Omron CX-Programmer project NewProject (CX-Programmer 9.73)

# PLC NewPLC1: CP1E N30

## Global symbols (name address type ; comment)
100.00 BOOL  ; C MERAH
100.01 BOOL  ; C MERAH BELOK
100.02 BOOL  ; B MERAH
100.03 BOOL  ; B MERAH BELOK
100.04 BOOL  ; D MERAH
100.05 BOOL  ; D MERAH BELOK
100.06 BOOL  ; D KUNING
100.07 BOOL  ; D KUNING BELOK
100.08 BOOL  ; ;
100.09 BOOL  ; A HIJAU BELOK
100.10 BOOL  ; A KUNING BELOK
100.11 BOOL  ; C KUNING
100.12 BOOL  ; C HIJAU
100.13 BOOL  ; C KUNING BELOK
100.14 BOOL  ; C HIJAU BELOK
100.15 BOOL  ; B KUNING
101.00 BOOL  ; B KUNING BELOK
101.01 BOOL  ; B HIJAU
101.02 BOOL  ; B HIJAU BELOK
101.03 BOOL  ; D HIJAU BELOK
101.04 BOOL  ; D HIJAU
101.05 BOOL  ; A KUNING
101.06 BOOL  ; A MERAH
101.07 BOOL  ; A MERAH BELOK
101.08 BOOL  ; A HIJAU KEDIP
101.09 BOOL  ; B HIJAU KEDIP
101.10 BOOL  ; C HIJAU KEDIP
101.11 BOOL  ; D HIJAU KEDIP
102.00 BOOL  ; A KEDIP
102.01 BOOL  ; B KEDIP
102.02 BOOL  ; C KEDIP
102.03 BOOL  ; D KEDIP

## Program NewProgram1 (cyclic task 0)

### Section Section1

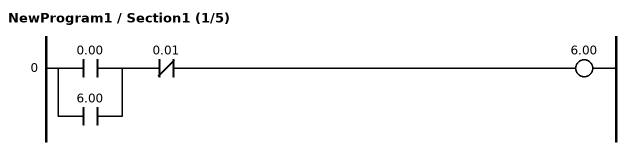
; rung 0
LD 0.00
OR 6.00
ANDNOT 0.01
OUT 6.00

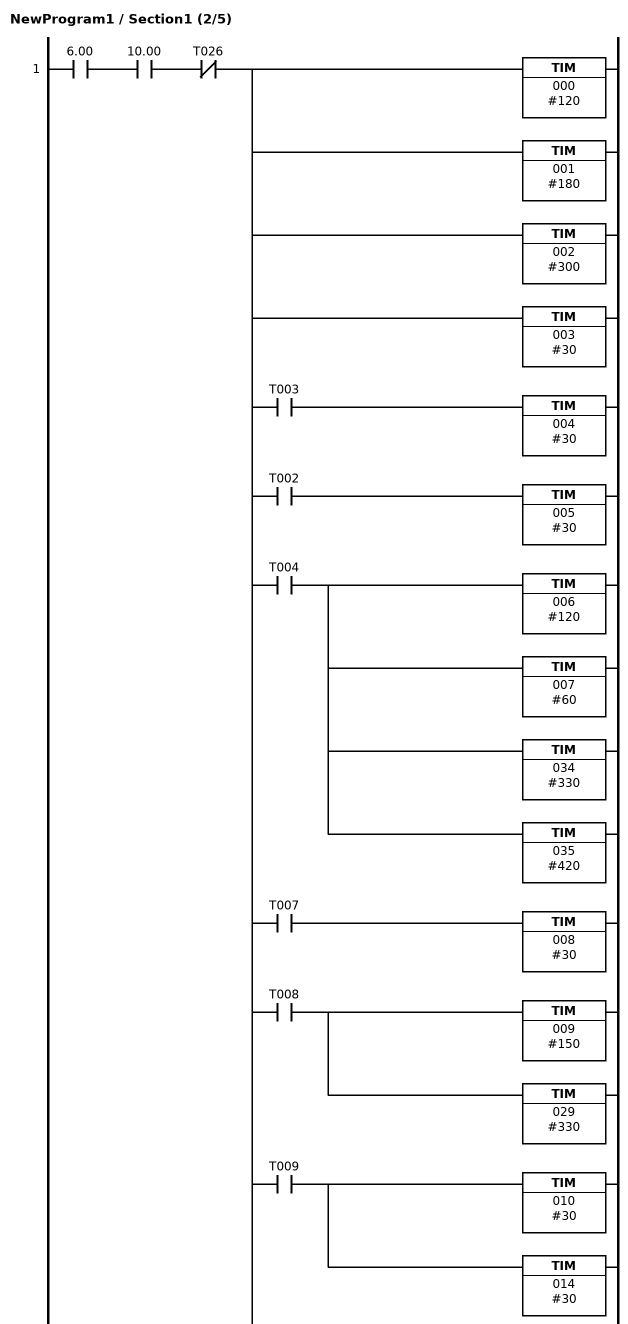

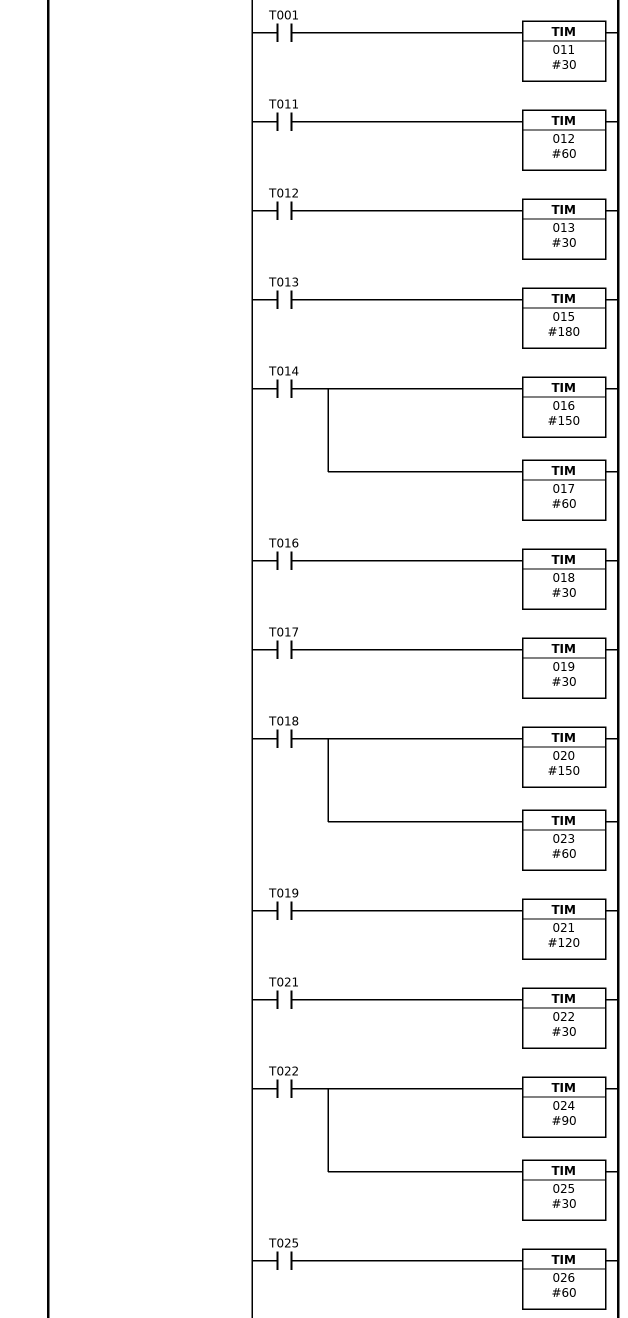

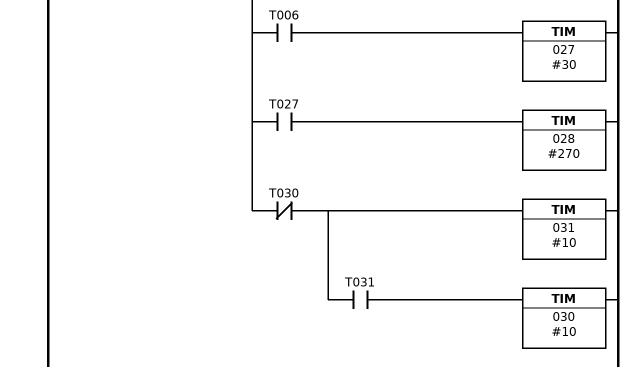
; rung 1
LD 6.00
AND 10.00
ANDNOT T026
OUT TR0
TIM 000 #120
TIM 001 #180
TIM 002 #300
TIM 003 #30
AND T003
TIM 004 #30
LD TR0
AND T002
TIM 005 #30
LD TR0
AND T004
TIM 006 #120
TIM 007 #60
TIM 034 #330
TIM 035 #420
LD TR0
AND T007
TIM 008 #30
LD TR0
AND T008
TIM 009 #150
TIM 029 #330
LD TR0
AND T009
TIM 010 #30
TIM 014 #30
LD TR0
AND T001
TIM 011 #30
LD TR0
AND T011
TIM 012 #60
LD TR0
AND T012
TIM 013 #30
LD TR0
AND T013
TIM 015 #180
LD TR0
AND T014
TIM 016 #150
TIM 017 #60
LD TR0
AND T016
TIM 018 #30
LD TR0
AND T017
TIM 019 #30
LD TR0
AND T018
TIM 020 #150
TIM 023 #60
LD TR0
AND T019
TIM 021 #120
LD TR0
AND T021
TIM 022 #30
LD TR0
AND T022
TIM 024 #90
TIM 025 #30
LD TR0
AND T025
TIM 026 #60
LD TR0
AND T006
TIM 027 #30
LD TR0
AND T027
TIM 028 #270
LD TR0
ANDNOT T030
TIM 031 #10
AND T031
TIM 030 #10

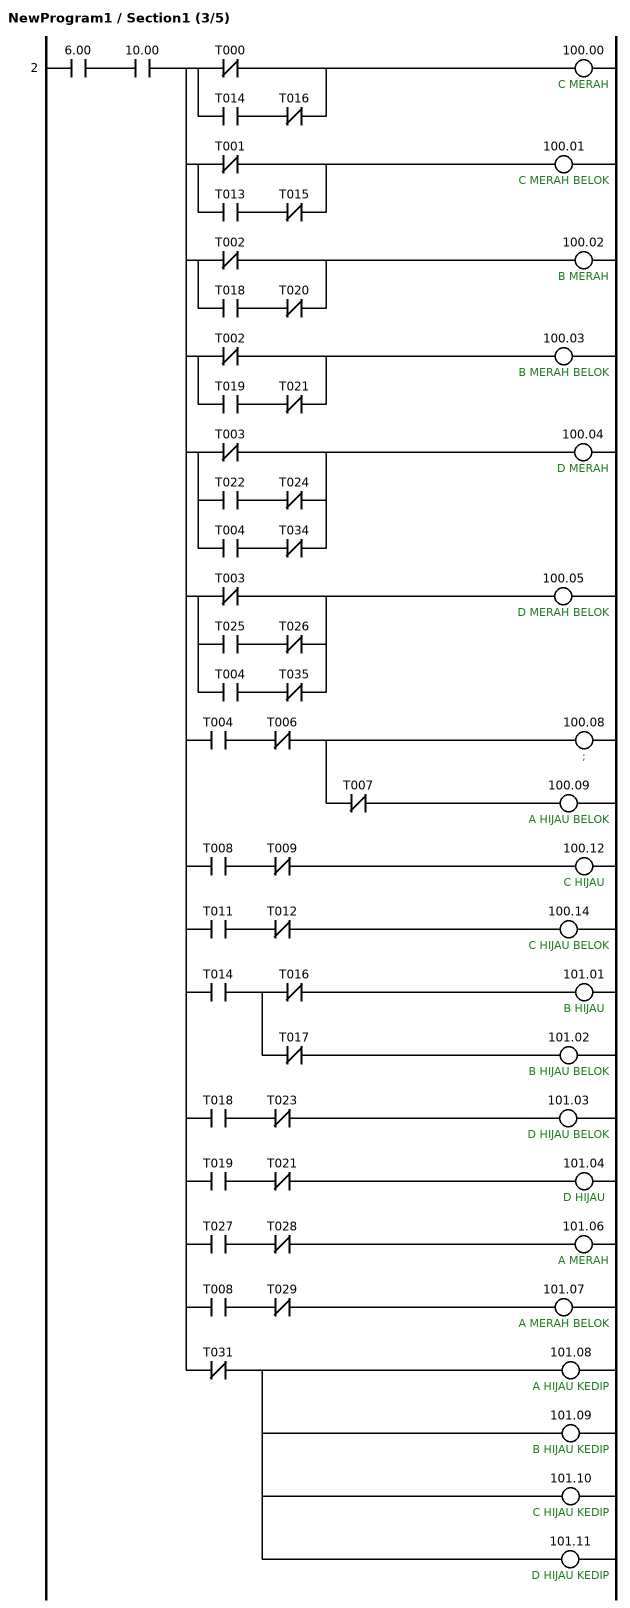
; rung 2
LD 6.00
AND 10.00
OUT TR0
LDNOT T000
LD T014
ANDNOT T016
ORLD
ANDLD
OUT 100.00  ; C MERAH
LD TR0
LDNOT T001
LD T013
ANDNOT T015
ORLD
ANDLD
OUT 100.01  ; C MERAH BELOK
LD TR0
LDNOT T002
LD T018
ANDNOT T020
ORLD
ANDLD
OUT 100.02  ; B MERAH
LD TR0
LDNOT T002
LD T019
ANDNOT T021
ORLD
ANDLD
OUT 100.03  ; B MERAH BELOK
LD TR0
LDNOT T003
LD T022
ANDNOT T024
ORLD
LD T004
ANDNOT T034
ORLD
ANDLD
OUT 100.04  ; D MERAH
LD TR0
LDNOT T003
LD T025
ANDNOT T026
ORLD
LD T004
ANDNOT T035
ORLD
ANDLD
OUT 100.05  ; D MERAH BELOK
LD TR0
AND T004
ANDNOT T006
OUT 100.08  ; ;
ANDNOT T007
OUT 100.09  ; A HIJAU BELOK
LD TR0
AND T008
ANDNOT T009
OUT 100.12  ; C HIJAU
LD TR0
AND T011
ANDNOT T012
OUT 100.14  ; C HIJAU BELOK
LD TR0
AND T014
OUT TR1
ANDNOT T016
OUT 101.01  ; B HIJAU
LD TR1
ANDNOT T017
OUT 101.02  ; B HIJAU BELOK
LD TR0
AND T018
ANDNOT T023
OUT 101.03  ; D HIJAU BELOK
LD TR0
AND T019
ANDNOT T021
OUT 101.04  ; D HIJAU
LD TR0
AND T027
ANDNOT T028
OUT 101.06  ; A MERAH
LD TR0
AND T008
ANDNOT T029
OUT 101.07  ; A MERAH BELOK
LD TR0
ANDNOT T031
OUT 101.08  ; A HIJAU KEDIP
OUT 101.09  ; B HIJAU KEDIP
OUT 101.10  ; C HIJAU KEDIP
OUT 101.11  ; D HIJAU KEDIP

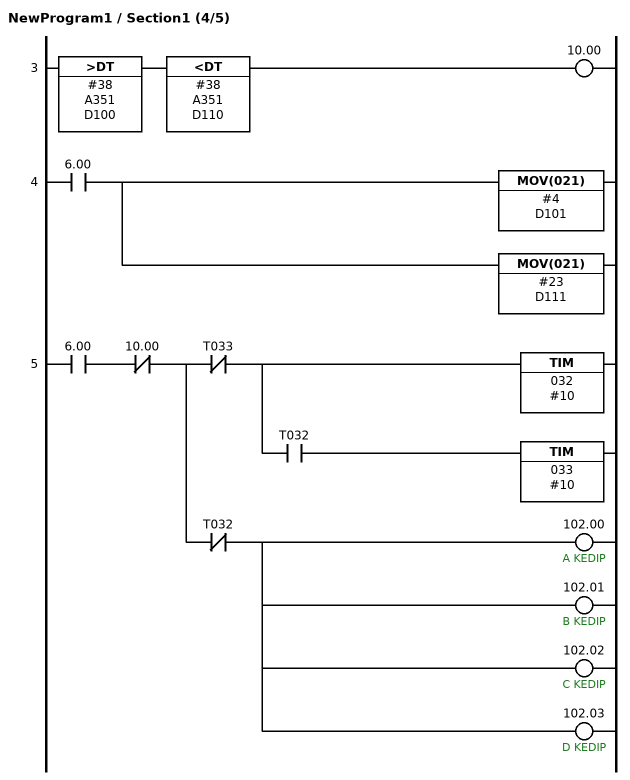
; rung 3
LD>DT(345) #38 A351 D100
AND<DT(343) #38 A351 D110
OUT 10.00
; rung 4
LD 6.00
MOV(021) #4 D101
MOV(021) #23 D111
; rung 5
LD 6.00
ANDNOT 10.00
OUT TR0
ANDNOT T033
TIM 032 #10
AND T032
TIM 033 #10
LD TR0
ANDNOT T032
OUT 102.00  ; A KEDIP
OUT 102.01  ; B KEDIP
OUT 102.02  ; C KEDIP
OUT 102.03  ; D KEDIP

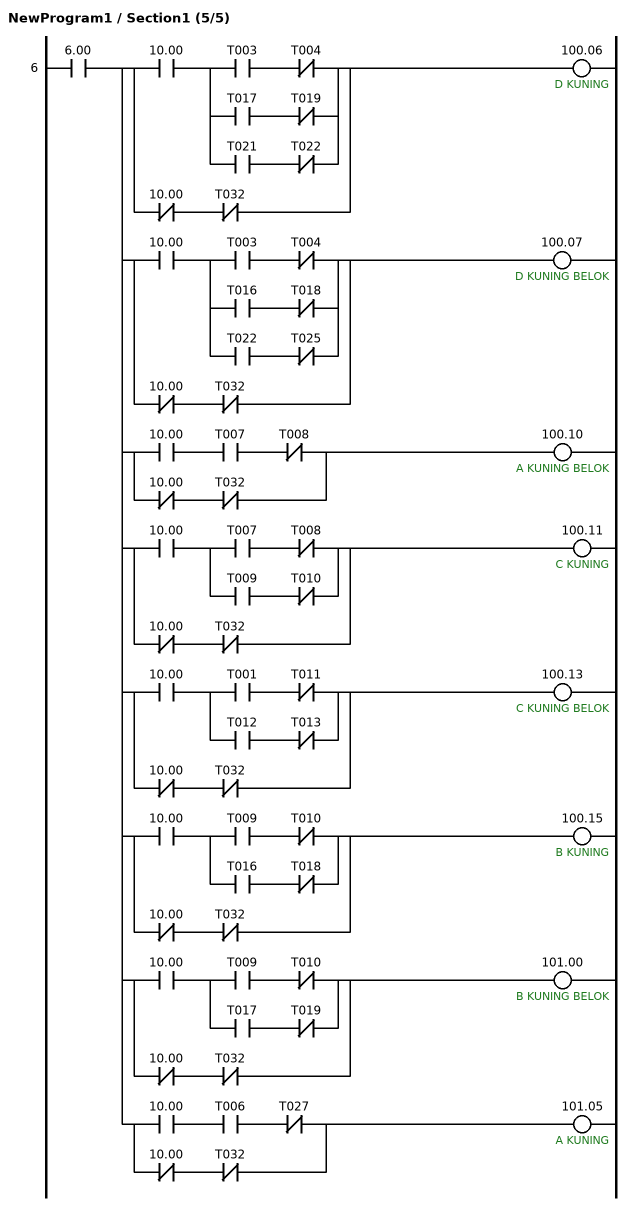
; rung 6
LD 6.00
OUT TR0
LD 10.00
LD T003
ANDNOT T004
LD T017
ANDNOT T019
ORLD
LD T021
ANDNOT T022
ORLD
ANDLD
LDNOT 10.00
ANDNOT T032
ORLD
ANDLD
OUT 100.06  ; D KUNING
LD TR0
LD 10.00
LD T003
ANDNOT T004
LD T016
ANDNOT T018
ORLD
LD T022
ANDNOT T025
ORLD
ANDLD
LDNOT 10.00
ANDNOT T032
ORLD
ANDLD
OUT 100.07  ; D KUNING BELOK
LD TR0
LD 10.00
AND T007
ANDNOT T008
LDNOT 10.00
ANDNOT T032
ORLD
ANDLD
OUT 100.10  ; A KUNING BELOK
LD TR0
LD 10.00
LD T007
ANDNOT T008
LD T009
ANDNOT T010
ORLD
ANDLD
LDNOT 10.00
ANDNOT T032
ORLD
ANDLD
OUT 100.11  ; C KUNING
LD TR0
LD 10.00
LD T001
ANDNOT T011
LD T012
ANDNOT T013
ORLD
ANDLD
LDNOT 10.00
ANDNOT T032
ORLD
ANDLD
OUT 100.13  ; C KUNING BELOK
LD TR0
LD 10.00
LD T009
ANDNOT T010
LD T016
ANDNOT T018
ORLD
ANDLD
LDNOT 10.00
ANDNOT T032
ORLD
ANDLD
OUT 100.15  ; B KUNING
LD TR0
LD 10.00
LD T009
ANDNOT T010
LD T017
ANDNOT T019
ORLD
ANDLD
LDNOT 10.00
ANDNOT T032
ORLD
ANDLD
OUT 101.00  ; B KUNING BELOK
LD TR0
LD 10.00
AND T006
ANDNOT T027
LDNOT 10.00
ANDNOT T032
ORLD
ANDLD
OUT 101.05  ; A KUNING

### Section END
; rung 0
END(001)